// TIA Portal V21 export
TYPE "AxixAS_DataOut_Type_v2.0"
   STRUCT
      oxCmdMotorForw : Bool;   // Inverter run enabled / Abilitazione marcia Avanti
      oxCmdMotorBack : Bool;   // Abilitazione marcia Indietro
      oxCmdBrake : Bool;   // Enable brake release / Comando stacco freno
      oxPosError { S7_SetPoint := 'True'} : Bool;   // Pursuit error / Allarme: Errore di inseguimento
      oxSincroError : Bool;   // Allarme: Sicro fuori tolleranza
      oxEndPos : Bool;   // Positioning terminated / Posizionamento terminato
      oxEndPosBig : Bool;   // Posizionamento Allargato terminato
      oxStopSpeed : Bool;   // Motor speed below low limit / Velocità motore = 0
      oxAccOnWork : Bool;   // Rampa Acc in atto
      oxDecOnWork : Bool;   // Rampa Dec in atto
      ofSpeedRequest : Real;   // Motor speed requested (mm/sec) / Velocita motore richiesta (mm/sec)
      ofEncMotorPos : Real;   // Motor encoder position (mm) / Posizione encoder motore (mm)
      ofMaxError : Real;   // Pursuit max error (mm) / Errore massimo di inseguimento (mm)
      ofSpaceStop : Real;   // Stop space requested from current position/speed (mm) / Spazio richiesto per fermata da posizione/velocità attuale (mm)
      ofSpaceLevRes : Real;   // Spazio richiesto per cambio velocità ricerca livello da posizione/velocità attuale (mm)
      ofSpaceStart : Real;   // Spazio richiesto per partenza da posizione/velocità attuale (mm)
      otTimeMove : Time;   // Tempo ultimo movimento
   END_STRUCT;
END_TYPE
